FUNCTION_BLOCK RASPBERRY_PI_TRIGGER_BUTTON
  {SET_ATTRIBUTE(OpcUa, DEVICE.SENSOR)}
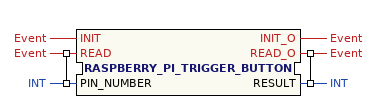
  EVENT_INPUT
    INIT;
    READ WITH PIN_NUMBER;
  END_EVENT
  EVENT_OUTPUT
    INIT_O;
    READ_O WITH RESULT;
  END_EVENT
  VAR_INPUT
    PIN_NUMBER : INT; {SET_ATTRIBUTE(OpcUa, Variable)}
  END_VAR
  VAR_OUTPUT
    RESULT : INT; {SET_ATTRIBUTE(OpcUa, Variable.RUN)}
  END_VAR
END_FUNCTION_BLOCK
